PROGRAM Medewerker
VAR
	state : MedewerkerToestand;
	
	orderCompleet : BOOL := FALSE;
	
	medewerkerTimer : TON;
END_VAR

CASE state OF
	MedewerkerToestand.wachtenOpKlant:
		// CODE
	MedewerkerToestand.klantHelpen:
		// CODE
		GVL.verfOrder[1] := GVL.merkVerf;
		GVL.verfOrder[2] := GVL.kleurVerf;
		GVL.verfOrder[3] := GVL.typeVerf;
		GVL.verfOrder[4] := GVL.hoeveelVerf;
		
		IF orderCompleet THEN
			state := MedewerkerToestand.verfMengen;
		END_IF
		
	MedewerkerToestand.verfMengen:
		medewerkerTimer(IN:= TRUE, PT:= T#7S); // Simulate the time it takes to click all buttons until scanning barcode
		// Blik onder kleurmachine zetten
		GVL.blikPresent := TRUE;
		// order aanklikken en starten
		GVL.opdrachtKnop := TRUE;
		GVL.startKnop := TRUE;
		IF medewerkerTimer.Q THEN
			// barcode scannen
		    GVL.barcodeBlik := 1234;
			GVL.opdrachtKnop := FALSE;
			GVL.startKnop := FALSE;
			IF kleurmachine.state = kleurmachineToestand.klaarMetToevoegen THEN
				GVL.blikPresent := FALSE;
				medewerkerTimer(IN:=FALSE);
				state := MedewerkerToestand.verfGeven;
			END_IF
			
		END_IF
		
	MedewerkerToestand.verfGeven:
		medewerkerTimer(IN:= TRUE, PT:= T#5S); // simulate giving can to customer
		IF medewerkerTimer.Q THEN
			GVL.verfAanKlantGegeven := TRUE;
			state := MedewerkerToestand.wachtenOpKlant;
		END_IF
		
		
END_CASE

END_PROGRAM

(* stored: Version 1.1.0.1, ProductVersion 3.1.4024.15
   POU Medewerker: Id {37e4aa0d-7777-400c-a8ca-388435fd5c5b}, SpecialFunc None *)
